SYSTEM AssemblyLine
  (* Version 1.0, 2025-03-21, AK123700 *)
  APPLICATION AssemblyLineApp
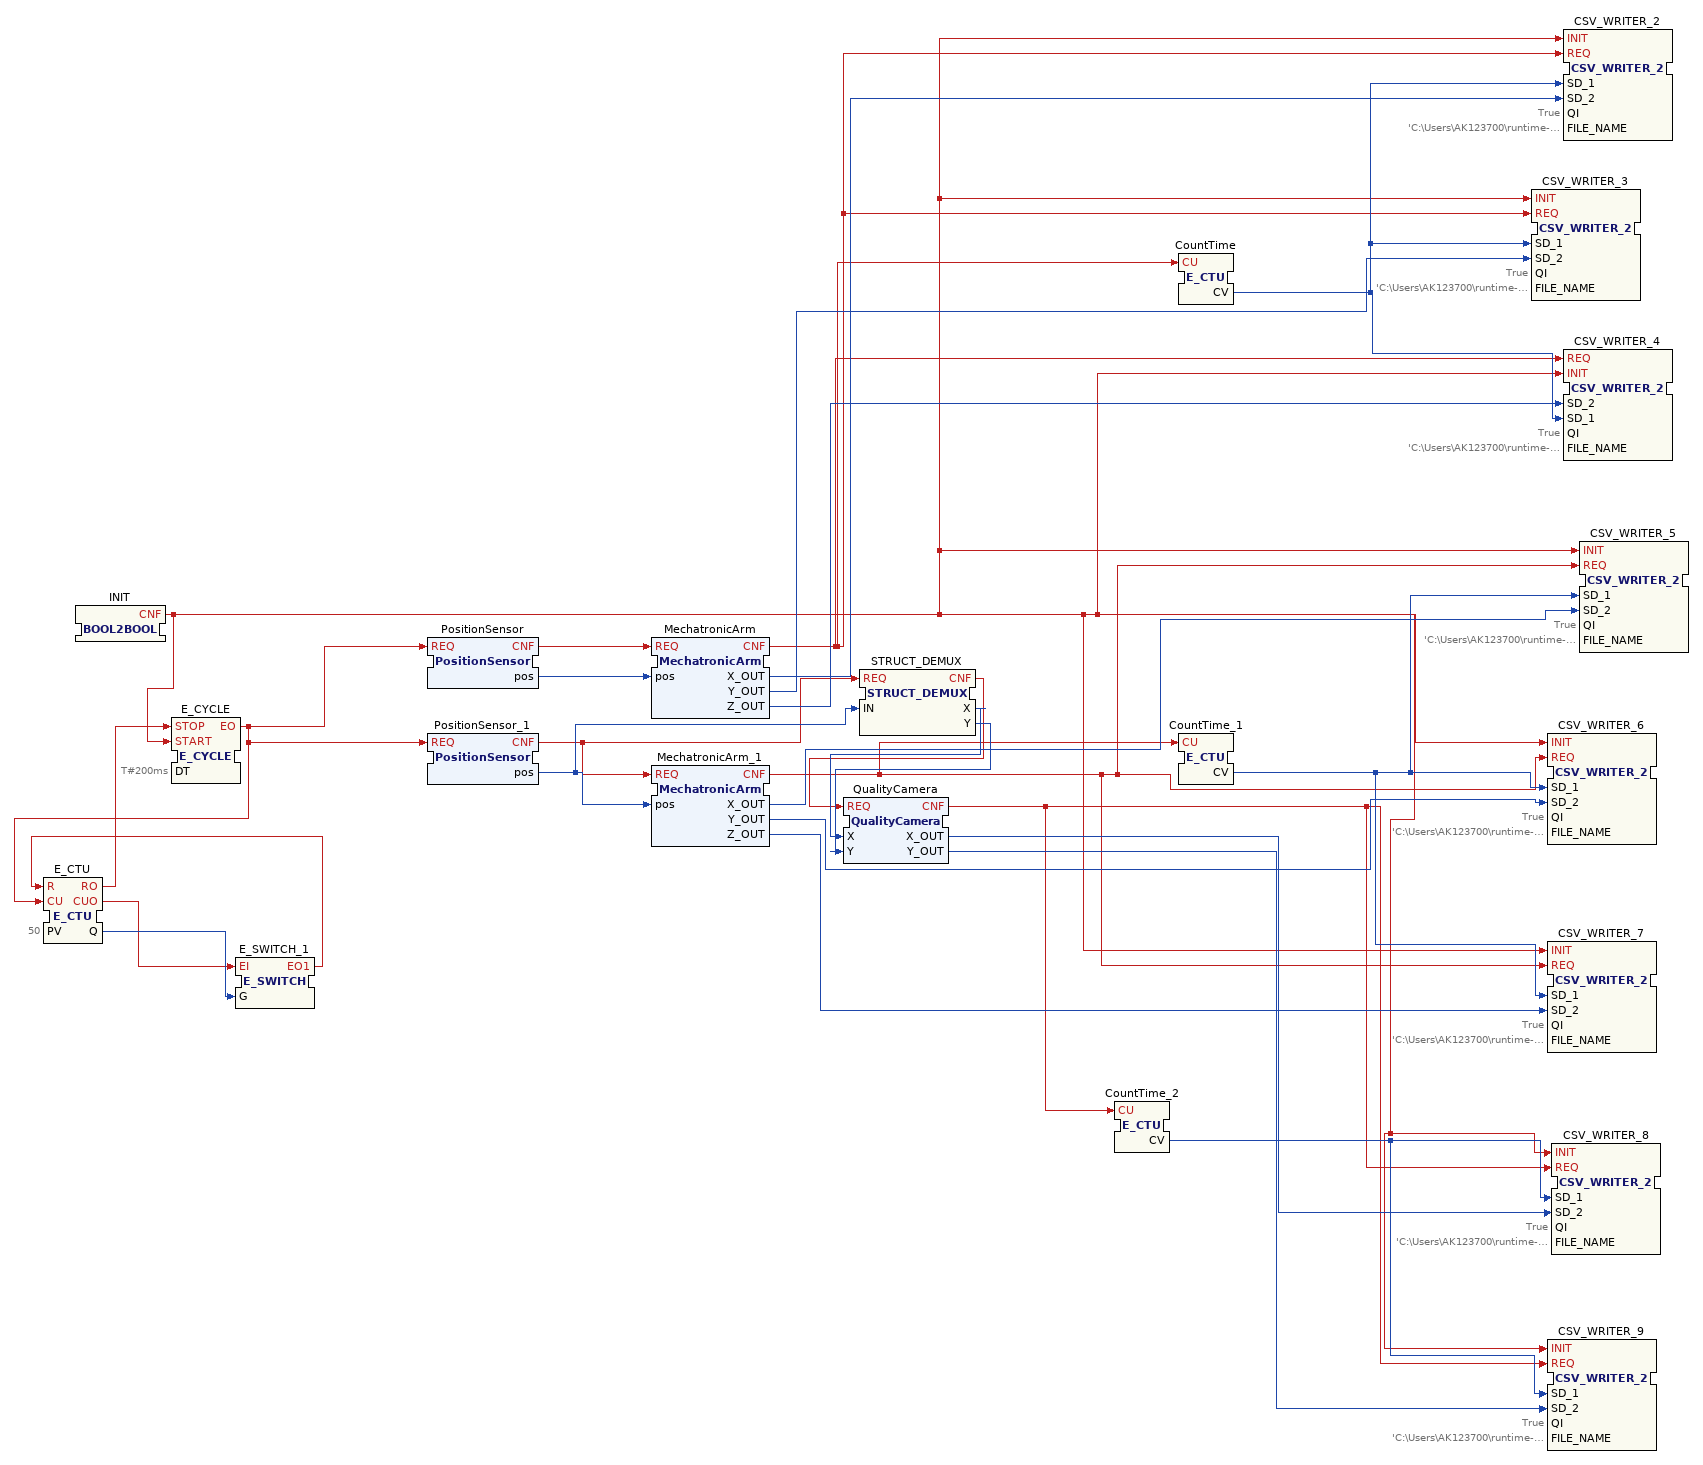
    FBS
      E_CYCLE : E_CYCLE(DT := T#200ms);
      CSV_WRITER_2 : CSV_WRITER_2(QI := True, FILE_NAME := 'C:\Users\AK123700\runtime-org.eclipse.fordiac.ide.product\AssemblyLineRepaired\traces\arm_x.csv');
      CountTime : E_CTU;
      E_CTU : E_CTU(PV := 50);
      INIT : BOOL2BOOL;
      E_SWITCH_1 : E_SWITCH;
      CSV_WRITER_3 : CSV_WRITER_2(QI := True, FILE_NAME := 'C:\Users\AK123700\runtime-org.eclipse.fordiac.ide.product\AssemblyLineRepaired\traces\arm_y.csv');
      CSV_WRITER_4 : CSV_WRITER_2(QI := True, FILE_NAME := 'C:\Users\AK123700\runtime-org.eclipse.fordiac.ide.product\AssemblyLineRepaired\traces\arm_z.csv');
      CSV_WRITER_5 : CSV_WRITER_2(QI := True, FILE_NAME := 'C:\Users\AK123700\runtime-org.eclipse.fordiac.ide.product\AssemblyLineRepaired\traces\arm1_x.csv');
      CSV_WRITER_6 : CSV_WRITER_2(QI := True, FILE_NAME := 'C:\Users\AK123700\runtime-org.eclipse.fordiac.ide.product\AssemblyLineRepaired\traces\arm1_y.csv');
      CSV_WRITER_7 : CSV_WRITER_2(QI := True, FILE_NAME := 'C:\Users\AK123700\runtime-org.eclipse.fordiac.ide.product\AssemblyLineRepaired\traces\arm1_z.csv');
      CountTime_1 : E_CTU;
      CountTime_2 : E_CTU;
      CSV_WRITER_8 : CSV_WRITER_2(QI := True, FILE_NAME := 'C:\Users\AK123700\runtime-org.eclipse.fordiac.ide.product\AssemblyLineRepaired\traces\camera_x.csv');
      CSV_WRITER_9 : CSV_WRITER_2(QI := True, FILE_NAME := 'C:\Users\AK123700\runtime-org.eclipse.fordiac.ide.product\AssemblyLineRepairedRepaired\traces\camery_y.csv');
      STRUCT_DEMUX : STRUCT_DEMUX; {SET_ATTRIBUTE(StructuredType, position)}
    END_FBS
    SUBAPPS
      PositionSensor : PositionSensor;
      MechatronicArm : MechatronicArm;
      QualityCamera : QualityCamera;
      PositionSensor_1 : PositionSensor;
      MechatronicArm_1 : MechatronicArm;
    END_SUBAPPS
    EVENT_CONNECTIONS
      E_CTU.RO TO E_CYCLE.STOP;
      INIT.CNF TO E_CYCLE.START;
      INIT.CNF TO CSV_WRITER_2.INIT;
      E_CTU.CUO TO E_SWITCH_1.EI;
      E_SWITCH_1.EO1 TO E_CTU.R;
      E_CYCLE.EO TO PositionSensor.REQ;
      PositionSensor.CNF TO MechatronicArm.REQ;
      MechatronicArm.CNF TO CountTime.CU;
      MechatronicArm.CNF TO CSV_WRITER_2.REQ;
      E_CYCLE.EO TO PositionSensor_1.REQ;
      INIT.CNF TO CSV_WRITER_3.INIT;
      MechatronicArm.CNF TO CSV_WRITER_3.REQ;
      MechatronicArm.CNF TO CSV_WRITER_4.REQ;
      INIT.CNF TO CSV_WRITER_4.INIT;
      E_CYCLE.EO TO E_CTU.CU;
      INIT.CNF TO CSV_WRITER_5.INIT;
      INIT.CNF TO CSV_WRITER_7.INIT;
      INIT.CNF TO CSV_WRITER_6.INIT;
      INIT.CNF TO CSV_WRITER_8.INIT;
      INIT.CNF TO CSV_WRITER_9.INIT;
      MechatronicArm_1.CNF TO CountTime_1.CU;
      QualityCamera.CNF TO CountTime_2.CU;
      MechatronicArm_1.CNF TO CSV_WRITER_5.REQ;
      MechatronicArm_1.CNF TO CSV_WRITER_6.REQ;
      MechatronicArm_1.CNF TO CSV_WRITER_7.REQ;
      QualityCamera.CNF TO CSV_WRITER_8.REQ;
      QualityCamera.CNF TO CSV_WRITER_9.REQ;
      STRUCT_DEMUX.CNF TO QualityCamera.REQ;
      PositionSensor_1.CNF TO STRUCT_DEMUX.REQ;
      PositionSensor_1.CNF TO MechatronicArm_1.REQ;
    END_CONNECTIONS
    DATA_CONNECTIONS
      CountTime.CV TO CSV_WRITER_2.SD_1;
      E_CTU.Q TO E_SWITCH_1.G;
      MechatronicArm.X_OUT TO CSV_WRITER_2.SD_2;
      STRUCT_DEMUX.X TO QualityCamera.X;
      STRUCT_DEMUX.Y TO QualityCamera.Y;
      CountTime.CV TO CSV_WRITER_3.SD_1;
      MechatronicArm.Y_OUT TO CSV_WRITER_3.SD_2;
      MechatronicArm.Z_OUT TO CSV_WRITER_4.SD_2;
      CountTime.CV TO CSV_WRITER_4.SD_1;
      CountTime_1.CV TO CSV_WRITER_6.SD_1;
      CountTime_1.CV TO CSV_WRITER_7.SD_1;
      CountTime_1.CV TO CSV_WRITER_5.SD_1;
      CountTime_2.CV TO CSV_WRITER_8.SD_1;
      CountTime_2.CV TO CSV_WRITER_9.SD_1;
      MechatronicArm_1.X_OUT TO CSV_WRITER_5.SD_2;
      MechatronicArm_1.Y_OUT TO CSV_WRITER_6.SD_2;
      MechatronicArm_1.Z_OUT TO CSV_WRITER_7.SD_2;
      QualityCamera.X_OUT TO CSV_WRITER_8.SD_2;
      QualityCamera.Y_OUT TO CSV_WRITER_9.SD_2;
      PositionSensor.pos TO MechatronicArm.pos;
      PositionSensor_1.pos TO MechatronicArm_1.pos;
      PositionSensor_1.pos TO STRUCT_DEMUX.IN;
    END_CONNECTIONS
  END_APPLICATION
  DEVICE FORTE_PC : FORTE_PC(MGR_ID := "localhost:61499" (* Device manager socket ID *))
    {SET_ATTRIBUTE(Profile, HOLOBLOC)}
    RESOURCE EMB_RES : EMB_RES
    END_RESOURCE
  END_DEVICE
  MAPPINGS
    AssemblyLineApp.CSV_WRITER_4 ON FORTE_PC.EMB_RES;
    AssemblyLineApp.CountTime_2 ON FORTE_PC.EMB_RES;
    AssemblyLineApp.E_CTU ON FORTE_PC.EMB_RES;
    AssemblyLineApp.INIT ON FORTE_PC.EMB_RES;
    AssemblyLineApp.CountTime_1 ON FORTE_PC.EMB_RES;
    AssemblyLineApp.CountTime ON FORTE_PC.EMB_RES;
    AssemblyLineApp.QualityCamera ON FORTE_PC.EMB_RES;
    AssemblyLineApp.CSV_WRITER_9 ON FORTE_PC.EMB_RES;
    AssemblyLineApp.PositionSensor ON FORTE_PC.EMB_RES;
    AssemblyLineApp.CSV_WRITER_8 ON FORTE_PC.EMB_RES;
    AssemblyLineApp.MechatronicArm ON FORTE_PC.EMB_RES;
    AssemblyLineApp.CSV_WRITER_3 ON FORTE_PC.EMB_RES;
    AssemblyLineApp.CSV_WRITER_2 ON FORTE_PC.EMB_RES;
    AssemblyLineApp.PositionSensor_1 ON FORTE_PC.EMB_RES;
    AssemblyLineApp.E_CYCLE ON FORTE_PC.EMB_RES;
    AssemblyLineApp.CSV_WRITER_5 ON FORTE_PC.EMB_RES;
    AssemblyLineApp.CSV_WRITER_6 ON FORTE_PC.EMB_RES;
    AssemblyLineApp.CSV_WRITER_7 ON FORTE_PC.EMB_RES;
    AssemblyLineApp.MechatronicArm_1 ON FORTE_PC.EMB_RES;
    AssemblyLineApp.E_SWITCH_1 ON FORTE_PC.EMB_RES;
    AssemblyLineApp.STRUCT_DEMUX ON FORTE_PC.EMB_RES;
  END_MAPPINGS
END_SYSTEM
